Fanuc TP program (LS listing): calc_pick_r.ls

/PROG  CALC_PICK_R
/ATTR
OWNER		= MNEDITOR;
COMMENT		= "TABLE PICK ANGLE";
PROG_SIZE	= 1669;
CREATE		= DATE 23-03-08  TIME 02:54:44;
MODIFIED	= DATE 23-11-16  TIME 00:32:34;
FILE_NAME	= CALC_PIC;
VERSION		= 0;
LINE_COUNT	= 61;
MEMORY_SIZE	= 2065;
PROTECT		= READ_WRITE;
TCD:  STACK_SIZE	= 0,
      TASK_PRIORITY	= 50,
      TIME_SLICE	= 0,
      BUSY_LAMP_OFF	= 0,
      ABORT_REQUEST	= 0,
      PAUSE_REQUEST	= 0;
DEFAULT_GROUP	= 1,*,*,*,*;
CONTROL_CODE	= 00000000 00000000;
/APPL
/APPL

AUTO_SINGULARITY_HEADER;
  ENABLE_SINGULARITY_AVOIDANCE   : TRUE;
/MN
   1:  --eg:CALCULATE THE PICK ANGLE OF THE CURRENT SLOT TO MAXIMIZE REACH AND
    :  PREVENT SINULARITY ;
   2:   ;
   3:  LBL[1:START] ;
   4:  --eg:MOVE ZERO INTO PICK OFFSET ANGLE ;
   5:  R[73:TABLE PK/DP R]=0    ;
   6:  PR[38,6:TABLE PCK OFFSET]=0    ;
   7:   ;
   8:  LBL[100:SELECT TEMPLATE] ;
   9:  --eg:CALCULATE ANGLE BASED ON TEMPLATE TYPE ;
  10:  IF R[1:ACTIVE TEMPLATE]=2,JMP LBL[200] ;
  11:  IF R[1:ACTIVE TEMPLATE]=3,JMP LBL[300] ;
  12:  IF R[1:ACTIVE TEMPLATE]=4,JMP LBL[400] ;
  13:  IF R[1:ACTIVE TEMPLATE]=5,JMP LBL[500] ;
  14:  IF R[1:ACTIVE TEMPLATE]=6,JMP LBL[600] ;
  15:  JMP LBL[9980] ;
  16:   ;
  17:  LBL[200:2" TEMPLATE] ;
  18:  IF (R[6:CUR PICK SLOT #]=40),R[73:TABLE PK/DP R]=((-5)) ;
  19:  IF (R[6:CUR PICK SLOT #]=52),R[73:TABLE PK/DP R]=(35) ;
  20:  IF (R[6:CUR PICK SLOT #]=64),R[73:TABLE PK/DP R]=(20) ;
  21:  IF (R[6:CUR PICK SLOT #]=90),R[73:TABLE PK/DP R]=((-10)) ;
  22:  IF (R[6:CUR PICK SLOT #]=162),R[73:TABLE PK/DP R]=((-45)) ;
  23:  IF (R[6:CUR PICK SLOT #]=94 OR R[6:CUR PICK SLOT #]=140),R[73:TABLE PK/DP R]=((-15)) ;
  24:  IF (R[6:CUR PICK SLOT #]=114),R[73:TABLE PK/DP R]=((-50)) ;
  25:  IF (R[6:CUR PICK SLOT #]=160),R[73:TABLE PK/DP R]=((-50)) ;
  26:  IF (R[6:CUR PICK SLOT #]=166),R[73:TABLE PK/DP R]=((-10)) ;
  27:  IF (R[6:CUR PICK SLOT #]=184),R[73:TABLE PK/DP R]=((-50)) ;
  28:  IF (R[6:CUR PICK SLOT #]=186),R[73:TABLE PK/DP R]=((-12)) ;
  29:  IF (R[6:CUR PICK SLOT #]=202),R[73:TABLE PK/DP R]=(15) ;
  30:  IF (R[6:CUR PICK SLOT #]=206),R[73:TABLE PK/DP R]=((-12)) ;
  31:  JMP LBL[9999] ;
  32:   ;
  33:  LBL[300:3" TEMPLATE] ;
  34:  IF (R[6:CUR PICK SLOT #]=34),R[73:TABLE PK/DP R]=(25) ;
  35:  IF (R[6:CUR PICK SLOT #]=42),R[73:TABLE PK/DP R]=(25) ;
  36:  IF (R[6:CUR PICK SLOT #]=76),R[73:TABLE PK/DP R]=((-50)) ;
  37:  IF (R[6:CUR PICK SLOT #]=90),R[73:TABLE PK/DP R]=((-45)) ;
  38:  IF (R[6:CUR PICK SLOT #]=94),R[73:TABLE PK/DP R]=(25) ;
  39:  IF (R[6:CUR PICK SLOT #]=102),R[73:TABLE PK/DP R]=(25) ;
  40:  JMP LBL[9999] ;
  41:   ;
  42:  LBL[400:4" TEMPLATE] ;
  43:  IF (R[6:CUR PICK SLOT #]=14),R[73:TABLE PK/DP R]=(25) ;
  44:  IF (R[6:CUR PICK SLOT #]=20),R[73:TABLE PK/DP R]=(25) ;
  45:  IF (R[6:CUR PICK SLOT #]=44),R[73:TABLE PK/DP R]=((-50)) ;
  46:  JMP LBL[9999] ;
  47:   ;
  48:  LBL[500:5" TEMPLATE] ;
  49:  IF (R[6:CUR PICK SLOT #]=36),R[73:TABLE PK/DP R]=((-50)) ;
  50:  JMP LBL[9999] ;
  51:   ;
  52:  LBL[600:6" TEMPLATE] ;
  53:  JMP LBL[9999] ;
  54:   ;
  55:  LBL[9980:TEMPLATE FAULT] ;
  56:  CALL TABLE_MSG(1) ;
  57:  UALM[11] ;
  58:  JMP LBL[100] ;
  59:   ;
  60:  LBL[9999:END] ;
  61:  PR[38,6:TABLE PCK OFFSET]=R[73:TABLE PK/DP R]    ;
/POS
/END
